FUNCTION_BLOCK PUBLIC ABSTRACT FB_Lamp IMPLEMENTS I_Subject, I_Lamp
VAR
	_ipObserver		: I_Observer;
END_VAR

METHOD PUBLIC Attach
VAR_INPUT
	ipObserver		: I_Observer;
END_VAR
IF (ipObserver = 0) THEN
	RETURN;
END_IF
_ipObserver := ipObserver;
END_METHOD

METHOD PUBLIC Detach
_ipObserver := 0;
END_METHOD

// Reduces the control value by 5 in the range of 10 to 100.
METHOD PUBLIC ABSTRACT DimDown
END_METHOD

// Increments the control value by 5 in the range of 10 to 100.
METHOD PUBLIC ABSTRACT DimUp
END_METHOD

// Sets the control value to 0.
METHOD PUBLIC ABSTRACT Off
END_METHOD

// Sets the control value to 100.
METHOD PUBLIC ABSTRACT On
END_METHOD

END_FUNCTION_BLOCK

(* stored: Version 1.1.0.1, ProductVersion 3.1.4024.11
   POU FB_Lamp: Id {97bddd59-a325-4ddf-9d6f-0fca30c94781}, SpecialFunc None
   Method Attach: Id {a057e1d6-aa74-421b-bd12-c7ff764a03a3}
   Method Detach: Id {cf3106ba-b1dc-4650-8704-0eedbfba2e23}
   Method DimDown: Id {8b7f88b1-e292-4c2a-aae1-75588f41b571}
   Method DimUp: Id {9fe37ea9-5990-4433-83f7-0a1847779f2a}
   Method Off: Id {f3e9436a-390c-4279-8082-229c248a628e}
   Method On: Id {1431a5df-dca8-4bc8-baee-a7920fa71212} *)
